{attribute 'OPC.UA.DA' := '1'}
FUNCTION_BLOCK Ed12dssShutter EXTENDS ShutterBase
VAR_INPUT
END_VAR
VAR_OUTPUT
END_VAR
VAR
	{attribute 'OPC.UA.DA' := '0'}
	_config : Ed12dssShutterConfig;		
	{attribute 'OPC.UA.DA' := '0'}
	IoEd12dssShutter : IoEd12dssShutter;
	
	{attribute 'OPC.UA.DA' := '0'}
	_deliverMessages : INT;
	
	ShutterIrisPositionMsg : STRING(255);
	
	{region 'Commands'}
	
	{attribute 'OPC.UA.DA' := '0'}
	_open : BOOL;
	{attribute 'OPC.UA.DA' := '0'}
	_close : BOOL;
	{attribute 'OPC.UA.DA' := '0'}			  		   
	_raiseProperties : BOOL;
			
	{endregion}		

	{attribute 'OPC.UA.DA' := '0'}
	_initDevice : BOOL;	
	
	{attribute 'OPC.UA.DA' := '0'}
	_itemScheduler : INT;	
	{attribute 'OPC.UA.DA' := '0'}
	_pulseGenerator : TON;			
	{attribute 'OPC.UA.DA' := '0'}
	_itemRaisedProperties : INT;

	{attribute 'OPC.UA.DA' := '0'}
	_itemCycling : INT;	
	
	{attribute 'OPC.UA.DA' := '0'}
	message : STRING;
	
	{attribute 'OPC.UA.DA' := '0'}
	_bCycling : BOOL;
		
END_VAR

// Init device
InitDevice();

CASE _deliverMessages OF			
	EFeedbackMsgEd12dss.ShutterIrisPositionMsg :	
		ShutterIrisPositionMsg := message;	
END_CASE
_deliverMessages := 0;
		
// Commands		
ManualOpen(_open);
ManualClose(_close);
Cycling(_bCycling);
RaisePropertiesChanged(_raiseProperties);

IF (NOT _open AND NOT _close AND NOT _raiseProperties) THEN
	MessageScheduler();
END_IF

METHOD PROTECTED Cycling
VAR_INPUT
	Execute : BOOL;
END_VAR
IF Execute THEN			
	IF _pulseGenerator.Q THEN
		_pulseGenerator(IN := FALSE, PT := T#10MS);
		
		CASE _itemCycling OF		
			0: _open := TRUE;
			   _close := FALSE;
				_itemCycling := 1;
				
			1: _open := FALSE;
			   _close := TRUE;
				_itemCycling := 0;
		
		END_CASE	
	ELSE
		_pulseGenerator(IN := TRUE, PT := T#500MS);	
	END_IF									
END_IF
END_METHOD

METHOD FB_init : BOOL
VAR_INPUT
	bInitRetains : BOOL; // if TRUE, the retain variables are initialized (warm start / cold start)
	bInCopyCode : BOOL;  // if TRUE, the instance afterwards gets moved into the copy code (online change)
	Config : Ed12dssShutterConfig;
END_VAR
IF Config.IsEnabled THEN
	_config := Config;
	
	SUPER^._shutterConfig.Name := Config.Name;
	SUPER^._shutterConfig.DeviceID := Config.DeviceID;
	SUPER^._shutterConfig.IsEnabled := Config.IsEnabled;
	SUPER^._shutterConfig.LogLevel := Config.LogLevel;
	
	SUPER^.Name := Config.Name;
	SUPER^.DeviceID := Config.DeviceID;	
	THIS^.Family := DeviceFamily.Shutter;
		
	_Logger.Information(_message.Reset().Append('Init ').
							Append('{').Append(TO_STRING(THIS^.Family)).Append('} - ').
							Append('{').Append(TO_STRING(Config.Name)).Append('}').ToString());																													
END_IF
END_METHOD

METHOD InitDevice
VAR_INPUT
END_VAR
IF NOT _initDevice THEN	
	_logger.Information(_message.Reset().
								Append(_config.Name).
								Append(' - Init device').ToString());
	
	THIS^.SetDone();
	_initDevice := TRUE;	
END_IF
END_METHOD

{attribute 'TcRpcEnable' := '1'}
METHOD PROTECTED ManualClose
VAR_INPUT
	Execute : BOOL;
END_VAR
IF Execute THEN
	_logger.Information(_message.Reset().
								Append(_config.Name).
								Append(' - ManualClose : ').ToString());								
	IoEd12dssShutter.OutputSwitchContactClosure := FALSE;
	_close := FALSE;		
END_IF
END_METHOD

{attribute 'TcRpcEnable' := '1'}
METHOD PROTECTED ManualOpen
VAR_INPUT
	Execute : BOOL;
END_VAR
IF Execute THEN
	_logger.Information(_message.Reset().
								Append(_config.Name).
								Append(' - ManualOpen : ').ToString());		
	IoEd12dssShutter.OutputSwitchContactClosure := TRUE;
	_open := FALSE;		
END_IF
END_METHOD

METHOD MessageScheduler
VAR_INPUT
END_VAR
CASE _itemScheduler OF
		0:  ShutterIrisPosition();		
			_itemScheduler := 0;		
END_CASE
END_METHOD

{attribute 'TcRpcEnable' := '1'}
METHOD RaisePropertiesChanged
VAR_INPUT
	Execute : BOOL;
END_VAR
IF Execute THEN		
	_raiseProperties := TRUE;	
	
	IF _pulseGenerator.Q THEN
		_pulseGenerator(IN := FALSE, PT := T#10MS);
		
		CASE _itemRaisedProperties OF		
			0: ShutterIrisPositionMsg := ' ';		   
				_itemRaisedProperties := 10;
				
			10: 
				_logger.Information(_message.Reset().
								    Append(_config.Name).
								    Append(' - RaisePropertiesChanged').ToString());
				_raiseProperties := FALSE;
				_itemRaisedProperties := 0;
		
		END_CASE
	
	ELSE
		_pulseGenerator(IN := TRUE, PT := T#200MS);	
	END_IF
		
END_IF
END_METHOD

METHOD ShutterIrisPosition 
VAR_INPUT
END_VAR
VAR 
	close : STRING := 'CLOSE';
	open : STRING := 'OPEN';
END_VAR
_deliverMessages := EFeedbackMsgEd12dss.ShutterIrisPositionMsg;

IF IoEd12dssShutter.OutputSwitchContactClosure THEN
	message := open; 	
ELSE
	message := close; 
END_IF
END_METHOD

END_FUNCTION_BLOCK

(* stored: Version 1.1.0.1, ProductVersion 3.1.4024.4
   POU Ed12dssShutter: Id {b22bcf16-8cd3-4c81-8172-4044d24b4355}, SpecialFunc None
   Folder Commands: Id {77124df0-12e3-4886-8fc5-edf9cbd1d3e4}
   Method Cycling: Id {057ed00b-db3f-4e25-afb0-58cefe5e1187}
   Method FB_init: Id {6da64d75-62be-4970-ab2c-00f2ffdbaad8}
   Method InitDevice: Id {e4177f0e-c528-41df-8121-eb6974e0e5cb}
   Method ManualClose: Id {3635d383-63a3-4f09-8ffa-ea4019c23ac2}
   Method ManualOpen: Id {3ff5bb0c-6767-4fc4-a432-5437c3f91236}
   Method MessageScheduler: Id {221baca8-9624-411a-98b0-b17726ff2748}
   Method RaisePropertiesChanged: Id {fbe6de41-9e46-4528-8c11-889e02f9d8f0}
   Method ShutterIrisPosition: Id {cc5ff000-e323-4928-a4fa-45e56c6c3690} *)
